{attribute 'linkalways'} 
{attribute 'no_explicit_call' := 'This FB is a CLASS and must be accessed using methods or properties'}
{attribute 'enable_dynamic_creation'}
FUNCTION_BLOCK _ETcVnOcrModelType EXTENDS EnumDatatypeBase
VAR
	localData : ETcVnOcrModelType;
	activeData : REFERENCE TO ETcVnOcrModelType;
	enumBaseDatatype : _ULINT(localData);
END_VAR

METHOD PRIVATE AddLocalEnumeration
VAR_INPUT
	Enumeration : T_MAXSTRING;
	Value : ETcVnOcrModelType;
END_VAR
AddEnumeration(Enumeration, Value);
END_METHOD

PROPERTY PUBLIC Address : PVOID
GET
Address := ADR(activeData);
END_GET
END_PROPERTY

METHOD PUBLIC ClearReference
VAR_INPUT
END_VAR
activeData REF= localData;
SetBaseDatatypeReference();
END_METHOD

METHOD PUBLIC Clone : I_Datatype
VAR
    pClone : POINTER TO _ETcVnOcrModelType;
END_VAR
pClone := __NEW(_ETcVnOcrModelType(InitialValue := Value));
Clone := pClone^;
END_METHOD

METHOD FB_init : BOOL
VAR_INPUT
	bInitRetains : BOOL; // if TRUE, the retain variables are initialized (warm start / cold start)
	bInCopyCode : BOOL;  // if TRUE, the instance afterwards gets moved into the copy code (online change)
	InitialValue : ETcVnOcrModelType;
END_VAR
localData := InitialValue;
AddBaseDatatype(enumBaseDatatype);
ClearReference();

AddLocalEnumeration('TCVN_OMT_NUMBERS', ETcVnOcrModelType.TCVN_OMT_NUMBERS);
AddLocalEnumeration('TCVN_OMT_NUMBERS_SC', ETcVnOcrModelType.TCVN_OMT_NUMBERS_SC);
AddLocalEnumeration('TCVN_OMT_UCLETTERS', ETcVnOcrModelType.TCVN_OMT_UCLETTERS);
AddLocalEnumeration('TCVN_OMT_NUMBERS_SC_UCLETTERS', ETcVnOcrModelType.TCVN_OMT_NUMBERS_SC_UCLETTERS);
END_METHOD

PROPERTY PUBLIC Identifier : T_MAXSTRING
GET
Identifier := 'ETcVnOcrModelType';
END_GET
END_PROPERTY

METHOD IsEnumeratorValueEqual : BOOL
VAR_INPUT
	Enumerator : I_KeyValueForwardEnumerator;
END_VAR
VAR
	storedValue : ETcVnOcrModelType;
END_VAR
IF NOT Enumerator.TryGet(storedValue) THEN
	RETURN;
END_IF

IsEnumeratorValueEqual := storedValue = activeData;
END_METHOD

METHOD PUBLIC MakeReferenceTo
VAR_INPUT
	ReferenceTarget : REFERENCE TO ETcVnOcrModelType;
END_VAR
activeData REF= ReferenceTarget;
SetBaseDatatypeReference();
END_METHOD

METHOD PROTECTED SetBaseDatatypeReference
VAR_INPUT
END_VAR
enumBaseDatatype.MakeReferenceTo(activeData);
END_METHOD

PROPERTY PUBLIC Size : UDINT
GET
Size := SIZEOF(activeData);
END_GET
END_PROPERTY

METHOD TryMakeReferenceTo : BOOL
VAR_INPUT
	Target : I_Datatype;
END_VAR
VAR
	targetAsEnum : I_EnumDatatype;
	pTargetData : POINTER TO ETcVnOcrModelType;
END_VAR
IF NOT Target.TryResolveAsEnumDatatype(targetAsEnum) THEN
	RETURN;
END_IF

IF targetAsEnum.Identifier <> Identifier THEN
	RETURN;
END_IF

pTargetData := Target.Address;
activeData REF= pTargetData^;
SetBaseDatatypeReference();
TryMakeReferenceTo := TRUE;
END_METHOD

PROPERTY PUBLIC Value : ETcVnOcrModelType
GET
Value := activeData;
END_GET
SET
activeData := Value;
END_SET
END_PROPERTY

END_FUNCTION_BLOCK

(* stored: Version 1.1.0.1
   POU _ETcVnOcrModelType: Id {8ac6ab4b-b376-4dd9-83cc-72d603942c12}, SpecialFunc None
   Folder Constructor: Id {5fd907ab-a064-4d87-9601-7afec1e3e720}
   Folder Private: Id {dfffcc45-c9a6-456f-a63e-980079891cff}
   Folder Protected: Id {a8ba8ce0-2f79-43b7-a8cb-9d72d1d903d0}
   Method AddLocalEnumeration: Id {cfafd4f5-4a03-42a0-8739-22d91f983408}
   Property Address: Id {c7c5396e-3d3a-422b-8a2a-8dd87a93a9a2}
   Get Get: Id {1cbe9b6d-b2c0-4577-b902-a7c931dfa93a}
   Method ClearReference: Id {a7c17fb0-49c4-438b-855d-390b1734c808}
   Method Clone: Id {1713bc29-2070-4c34-864e-dc982138405e}
   Method FB_init: Id {c18fa77b-692f-47ed-a6e7-03dd33eb1f78}
   Property Identifier: Id {9fda9600-e55b-4a3f-9884-3608c0dddcfc}
   Get Get: Id {a55b3737-7b5f-479d-aaa7-f2d0c33a0bd9}
   Method IsEnumeratorValueEqual: Id {08b5025d-0f5b-450d-8856-825985d6dcfd}
   Method MakeReferenceTo: Id {41b79f0f-9344-483c-ac61-2f0cd0fe1d94}
   Method SetBaseDatatypeReference: Id {0337700f-9162-427e-8ddd-e93d7f674bec}
   Property Size: Id {99aadd11-8ed4-468d-bfee-980f438d005e}
   Get Get: Id {d79e2e88-3edc-4b72-8764-174508ef21f0}
   Method TryMakeReferenceTo: Id {f6e0926c-8de7-4ba7-a057-637a388ccc11}
   Property Value: Id {dd979463-1722-4820-bb15-59fa5d3f546c}
   Get Get: Id {634d4ce5-0ff8-4793-bf75-35898723f74a}
   Set Set: Id {1db4a661-69b7-4724-a38b-ed8402223d15} *)
